(*
SPDX-FileCopyrightText: © 2026 Oleksandr Tiutyk <trofimich@gmail.com>
SPDX-License-Identifier: MIT
License: https://opensource.org/license/mit
*)

(*!
<summary>Provides object address conversion, memory-area classification and explicit dynamic memory release.</summary>
<description>
Release requires a live allocation owned by the caller. These helpers do not log object disposal; object
FB_init, FB_exit and FB_reinit implementations must not create or raise exceptions. TryRelease methods contain
exceptions and clear the supplied address/reference on exceptional failure; this does not clear other aliases.
</description>
*)

{attribute 'no_explicit_call' := 'Direct call is not allowed'}
PROGRAM Memory
VAR CONSTANT
	//!<summary>
	//! Null data address used to detect an unassigned buffer pointer; a non-null address alone does not prove
	//! validity or capacity.
	//! </summary>
	NULL_ADDRESS : PVOID := 0;
END_VAR
VAR
	{attribute 'hide'} 
	_ClassName : STRING := __POUNAME();
END_VAR

{attribute 'monitoring' := 'call'}
PROPERTY ClassName : REFERENCE TO STRING
GET
ClassName REF= _ClassName;
END_GET
END_PROPERTY

(*!
<summary>Returns the borrowed address of a live FB instance; does not transfer ownership.</summary>
<description>
Returns 0 for a null interface or failed conversion. Does not validate lifetime.
</description>
*)

METHOD GetAddressFromInterface : PVOID
VAR_INPUT
	interfaceInstance : __SYSTEM.IQueryInterface; 
END_VAR
VAR
	instancePointer : POINTER TO BYTE;
END_VAR
IF interfaceInstance <> 0 AND_THEN __QUERYPOINTER(interfaceInstance, instancePointer) THEN
	GetAddressFromInterface := instancePointer;
END_IF
END_METHOD

(*!
<summary>Checks whether the specified memory range resides in stack memory.</summary>
<description>
Returns TRUE if the memory area classification is Unknown (which includes stack variables),
or FALSE if the memory is in static or dynamic PLC areas. Returns FALSE for null dataAddress.
</description>
*)
METHOD IsStackData : BOOL
VAR_INPUT
	dataAddress : PVOID;
	dataSize : UDINT := 1;
END_VAR
IF dataAddress = 0 THEN
	IsStackData := FALSE;
	RETURN;
END_IF

IsStackData := Tc2_System.F_CheckMemoryArea(
	pData := dataAddress,
	nSize := dataSize
) = E_TcMemoryArea.Unknown;
END_METHOD

(*!
<summary>Classifies the memory area only; does not prove allocation lifetime or ownership.</summary>
*)

METHOD IsDynamicData : BOOL
VAR_INPUT
	dataAddress : PVOID;
	dataSize : UDINT := 1;
END_VAR
IsDynamicData := Tc2_System.F_CheckMemoryArea(
	pData := dataAddress,
	nSize := dataSize
) = E_TcMemoryArea.Dynamic;
END_METHOD

(*!
<summary>Provides the library namespace used in diagnostics.</summary>
<description>
Borrowed read-only reference to the compiler-initialized library namespace; no ownership transfer.
</description>
*)
{attribute 'monitoring' := 'call'}
PROPERTY NamespaceName : REFERENCE TO STRING
GET
NamespaceName REF= CurrentNamespace.Name;
END_GET
END_PROPERTY

(*!
<summary>
Caller must own a live allocation. Registered auto-disposed objects are released only by their manager.
</summary>
<description>
Object FB_exit implementations must not raise exceptions. This method does not log disposal. Returns FALSE for
null/non-dynamic addresses without changing them. Catches exceptions and returns FALSE with address set to
zero to prevent reuse of a possibly partially destroyed allocation. TRUE means deletion completed with no terminal allocation failure observed.
Cleanup still runs with the latch set. A completed deletion clears the address even when returning FALSE. FALSE after
an exception does not guarantee that memory was freed. Other aliases are not cleared and must not be used or
deleted after a destruction failure. Terminal allocation state is preserved.
</description>
*)

METHOD TryReleaseDynamicMemory : BOOL
VAR_IN_OUT
	address : POINTER TO BYTE;	
END_VAR
VAR_INPUT
	isObject : BOOL;
END_VAR
VAR
	objectPointer : POINTER TO Object;
END_VAR
__TRY
	IF address = 0 OR_ELSE NOT Memory.IsDynamicData(dataAddress := address, dataSize := 1) THEN
		RETURN;
	END_IF

	IF isObject THEN
		objectPointer := address;
		
		__DELETE(objectPointer);
		address := 0;
	ELSE
		__DELETE(address);
	END_IF

	TryReleaseDynamicMemory := NOT DynamicMemoryManager.HasAllocationFailed;
__CATCH
	address := 0;
	TryReleaseDynamicMemory := FALSE;
__ENDTRY
END_METHOD

(*!
<summary>Caller must own the object; registered auto-disposed objects are released only by their manager.</summary>
<description>
Attempts cleanup even if SelfAddress contained a terminal allocation failure. A completed deletion clears
the interface even when the allocation latch forces FALSE. Returns FALSE for null or non-dynamic objects.
A non-dynamic reference remains unchanged. Clears instance after successful deletion or when the release helper clears the address on an
exception. Exceptions from obtaining SelfAddress are also caught with instance cleared. Other aliases remain
the caller's responsibility; FALSE does not guarantee an intact object or successful deallocation.
</description>
*)

METHOD TryReleaseDynamicObject : BOOL
VAR_IN_OUT
	instance : IObject;	
END_VAR
VAR
	objectPointer : POINTER TO Object;
END_VAR
__TRY
	IF instance = 0 THEN
		RETURN;
	END_IF
		
	objectPointer := instance.SelfAddress;

	TryReleaseDynamicObject := TryReleaseDynamicMemory(address := objectPointer, isObject := TRUE);

	IF TryReleaseDynamicObject OR_ELSE objectPointer = 0 THEN
		instance := 0;
	END_IF	
__CATCH
	instance := 0;
	TryReleaseDynamicObject := FALSE;
__ENDTRY
END_METHOD

END_PROGRAM

(* stored: Version 1.1.0.1
   POU Memory: Id {cb04704d-a05c-4735-b40b-67a92f3f86d5}, SpecialFunc None
   Property ClassName: Id {f0cb7e04-3fa7-438c-9fb8-38f358e717d9}
   Get Get: Id {9465e911-db84-4abe-a766-2f2cfe6e21d4}
   Method GetAddressFromInterface: Id {6158ab88-0c76-435a-bca8-37fff74aaa20}
   Method IsStackData: Id {b9f5f780-4a0e-4ae7-b4ae-b7ce9da8477c}
   Method IsDynamicData: Id {4c5114c7-cc73-448a-9f8f-fa67bfde37e3}
   Property NamespaceName: Id {5aeb5d90-3cbf-4d4b-8537-6b3b6ccb7bea}
   Get Get: Id {464e75ad-f0ba-4929-8b1e-1713c91d4754}
   Method TryReleaseDynamicMemory: Id {5fe5bc2a-b608-418e-9ff0-e9c1a91c92f5}
   Method TryReleaseDynamicObject: Id {1a29f8e6-f929-40c9-bee2-ed6219c50a45} *)
